TYPE PID_Parameter_Strukt :
STRUCT
	Kp :		REAL;
	Ti :		REAL;
	Td :		REAL;
	N :			REAL;
	ARW :		BOOL;
	Tr :		REAL;
	umin :		REAL;
	umax :		REAL;
END_STRUCT
END_TYPE

(* stored: Version 1.1.0.1, ProductVersion 3.1.4024.13
   DUT PID_Parameter_Strukt: Id {47b3e65c-c6b3-45be-8505-0062d15a7880} *)
